Yaskawa INFORM job: 123.JBI

/JOB
//NAME 123
//POS
///NPOS 0,0,0,0
//INST
///DATE 2014/11/02 19:10
///ATTR 0,0,0,0,0,0,0,0,0,0,0,0,0,1,0,0
///FRAME BASE
NOP
END
